PROGRAM LOAD_LASER
VAR_INPUT

END_VAR

VAR
	TMR_DELAY: TON;
	TMR1:TON;
	TMR_STOPPER_A: TON;
	TMR_STOPPER_B: TON;
END_VAR

CASE SORTER_VAR.I_CASE OF
0: //standby near lotbox
	IF SORTER_VAR.ACTIVE_ID=6 THEN
		SORTER_VAR.ACTIVE_ID:=1;
	END_IF
	CASE SORTER_VAR.I_CURRENT_TRANSACTION.TRANSPORT_INDEX OF
		2 : LASER_MOVE(STEP_DATA_1:=SORTER_VAR.I_CURRENT_TRANSACTION.STATION_NUMBER_LOAD,
				STEP_DATA_2:=3,
				STEP_DATA_3:=SORTER_VAR.I_CURRENT_TRANSACTION.JIG_INDEX_LOAD,
				STEP_DATA_4:=0,
				STEP_DATA_5:=1);
				SORTER_VAR.O_STOPPER_TRANSFER_B:=FALSE;
		1 : LASER_MOVE(STEP_DATA_1:=SORTER_VAR.I_CURRENT_TRANSACTION.STATION_NUMBER_LOAD,
				STEP_DATA_2:=3,
				STEP_DATA_3:=SORTER_VAR.I_CURRENT_TRANSACTION.JIG_INDEX_LOAD,
				STEP_DATA_4:=1,
				STEP_DATA_5:=0);
				SORTER_VAR.O_STOPPER_TRANSFER_A:=FALSE;
	END_CASE			
	SORTER_VAR.O_VACUUM_On:=FALSE;
	SORTER_VAR.O_VACUUM_OFF:=FALSE;	
	
			
1: //standby near lotbox
	
	IF SORTER_VAR.ACTIVE_ID=6 THEN
		SORTER_VAR.ACTIVE_ID:=1;
	END_IF
		LASER_MOVE(STEP_DATA_1:=SORTER_VAR.I_CURRENT_TRANSACTION.STATION_NUMBER_LOAD,
				STEP_DATA_2:=4,
				STEP_DATA_3:=SORTER_VAR.I_CURRENT_TRANSACTION.JIG_INDEX_LOAD,
				STEP_DATA_4:=0,
				STEP_DATA_5:=0);

		CASE SORTER_VAR.I_CURRENT_TRANSACTION.TRANSPORT_INDEX OF
		1:
			SORTER_VAR.I_LOADING_DONE_A:=FALSE;
		
		2:
			SORTER_VAR.I_LOADING_DONE_B:=FALSE;
	END_CASE
	
				
2://vacuum position 
	IF SORTER_VAR.ACTIVE_ID=6 THEN
		SORTER_VAR.ACTIVE_ID:=1;
	END_IF
	SORTER_VAR.I_CASE:=SORTER_VAR.I_CASE+1;
	(*LASER_MOVE(STEP_DATA_1:=SORTER_VAR.I_CURRENT_TRANSACTION.STATION_NUMBER_LOAD,
				STEP_DATA_2:=4,
				STEP_DATA_3:=SORTER_VAR.I_CURRENT_TRANSACTION.JIG_INDEX_LOAD,
				STEP_DATA_4:=0,
				STEP_DATA_5:=0);
	IF SORTER_VAR.ACTIVE_ID=3 THEN
		SORTER_VAR.O_VACUUM_ON:=TRUE;
		SORTER_VAR.O_VACUUM_OFF:=FALSE;	
	END_IF
	*)

3://vacuum position 
	IF SORTER_VAR.ACTIVE_ID=6 THEN
		SORTER_VAR.ACTIVE_ID:=1; 
	END_IF
	SORTER_VAR.I_CASE:=SORTER_VAR.I_CASE+1;
(*
		LASER_MOVE(STEP_DATA_1:=SORTER_VAR.I_CURRENT_TRANSACTION.STATION_NUMBER_LOAD,
				STEP_DATA_2:=4,
				STEP_DATA_3:=SORTER_VAR.I_CURRENT_TRANSACTION.JIG_INDEX_LOAD,
				STEP_DATA_4:=0,
				STEP_DATA_5:=0);
*)
4://vacuum position 
	IF SORTER_VAR.ACTIVE_ID=6 THEN
		SORTER_VAR.ACTIVE_ID:=1;
	END_IF
	SORTER_VAR.O_VACUUM_ON:=TRUE;
	SORTER_VAR.O_VACUUM_OFF:=FALSE;
	//CHECK JIG LASER PRESENCE	
LASER_MOVE(STEP_DATA_1:=SORTER_VAR.I_CURRENT_TRANSACTION.STATION_NUMBER_LOAD,
				STEP_DATA_2:=4,
				STEP_DATA_3:=SORTER_VAR.I_CURRENT_TRANSACTION.JIG_INDEX_LOAD,
				STEP_DATA_4:=0,
				STEP_DATA_5:=0);
(*		
	IF  SORTER_VAR.O_VACUUM_ON THEN
		TMR1(IN:=TRUE,PT:=T#2S);
		IF TMR1.Q THEN
			IF  SORTER_VAR.I_VACUUM_ON AND SORTER_VAR.O_VACUUM_ON THEN
				SORTER_VAR.JIG_LASER_PRESENCE :=TRUE;
				
				LASER_MOVE(STEP_DATA_1:=7,
				STEP_DATA_2:=4,
				STEP_DATA_3:=SORTER_VAR.I_CURRENT_TRANSACTION.JIG_INDEX_LOAD,
				STEP_DATA_4:=0,
				STEP_DATA_5:=0);
			ELSE
				SORTER_VAR.JIG_LASER_PRESENCE :=FALSE;	
				LASER_MOVE(STEP_DATA_1:=SORTER_VAR.I_CURRENT_TRANSACTION.STATION_NUMBER_LOAD,
				STEP_DATA_2:=2,
				STEP_DATA_3:=SORTER_VAR.I_CURRENT_TRANSACTION.JIG_INDEX_LOAD,
				STEP_DATA_4:=0,
				STEP_DATA_5:=0);
				
				LASER_MOVE(STEP_DATA_1:=SORTER_VAR.I_CURRENT_TRANSACTION.STATION_NUMBER_LOAD,
				STEP_DATA_2:=1,
				STEP_DATA_3:=SORTER_VAR.I_CURRENT_TRANSACTION.JIG_INDEX_LOAD,
				STEP_DATA_4:=0,
				STEP_DATA_5:=0);
				
				TMR_DELAY(IN:=TRUE,PT:=T#2S);
				IF TMR_DELAY.Q THEN
					FLAG_VAR.ALLOW_EXECUTE_LOAD_LASER:=FALSE;
					SORTER_VAR.I_CURRENT_TRANSACTION.JIG_INDEX_LOAD:=SORTER_VAR.I_CURRENT_TRANSACTION.JIG_INDEX_LOAD+0;
					SORTER_VAR.I_CASE:=0;
					TMR1(IN:=FALSE);
					SORTER_VAR.O_VACUUM_ON:=FALSE;
					SORTER_VAR.O_VACUUM_OFF:=FALSE;
				END_IF
			END_IF
		END_IF 
	END_IF
*)
				

5://vacuum position 
	IF SORTER_VAR.ACTIVE_ID=6 THEN
		SORTER_VAR.ACTIVE_ID:=1;
	END_IF

	LASER_MOVE(STEP_DATA_1:=SORTER_VAR.I_CURRENT_TRANSACTION.STATION_NUMBER_LOAD,//9,
				STEP_DATA_2:=2,
				STEP_DATA_3:=SORTER_VAR.I_CURRENT_TRANSACTION.JIG_INDEX_LOAD,
				STEP_DATA_4:=0,
				STEP_DATA_5:=0);

6://gripping position
	IF SORTER_VAR.ACTIVE_ID=6 THEN
		SORTER_VAR.ACTIVE_ID:=1;
	END_IF

	LASER_MOVE(STEP_DATA_1:=SORTER_VAR.I_CURRENT_TRANSACTION.TRANSPORT_INDEX+5,
				STEP_DATA_2:=1,
				STEP_DATA_3:=12,
				STEP_DATA_4:=0,
				STEP_DATA_5:=0);


7://placing onto LASER transport
	IF SORTER_VAR.ACTIVE_ID=6 THEN
		SORTER_VAR.ACTIVE_ID:=1;
	END_IF
	LASER_MOVE(STEP_DATA_1:=SORTER_VAR.I_CURRENT_TRANSACTION.TRANSPORT_INDEX+5,
				STEP_DATA_2:=1,
				STEP_DATA_3:=11,
				STEP_DATA_4:=0,
				STEP_DATA_5:=0);

8://placing onto LASER transport
	IF SORTER_VAR.ACTIVE_ID=6 THEN
		SORTER_VAR.ACTIVE_ID:=1;
	END_IF
	
	LASER_MOVE(STEP_DATA_1:=SORTER_VAR.I_CURRENT_TRANSACTION.TRANSPORT_INDEX+5,
				STEP_DATA_2:=1,
				STEP_DATA_3:=11,
				STEP_DATA_4:=0,
				STEP_DATA_5:=0);
	(*IF SORTER_VAR.ACTIVE_ID=3 THEN
		SORTER_VAR.O_VACUUM_On:=FALSE;
		SORTER_VAR.O_VACUUM_OFF:=TRUE;	
	END_IF
	*)
	
9://homing
	IF SORTER_VAR.ACTIVE_ID=6 THEN
		SORTER_VAR.ACTIVE_ID:=1;
	END_IF
	
			LASER_MOVE(STEP_DATA_1:=SORTER_VAR.I_CURRENT_TRANSACTION.TRANSPORT_INDEX+5,
				STEP_DATA_2:=0,
				STEP_DATA_3:=11,
				STEP_DATA_4:=0,
				STEP_DATA_5:=0);
	(*
	IF SORTER_VAR.I_VACUUM_ON THEN
		LASER_MOVE(STEP_DATA_1:=SORTER_VAR.I_CURRENT_TRANSACTION.TRANSPORT_INDEX+5,
				STEP_DATA_2:=1,
				STEP_DATA_3:=11,
				STEP_DATA_4:=0,
				STEP_DATA_5:=0);
	ELSE
		SORTER_VAR.O_VACUUM_On:=FALSE;
		SORTER_VAR.O_VACUUM_OFF:=TRUE;
	END_IF	
	*)			
10://pusH LASER transport
	IF SORTER_VAR.ACTIVE_ID=6 THEN
		SORTER_VAR.ACTIVE_ID:=1;
	END_IF
	SORTER_VAR.O_VACUUM_OFF:=FALSE;
	CASE SORTER_VAR.I_CURRENT_TRANSACTION.TRANSPORT_INDEX OF
		2 :
			IF NOT SORTER_VAR.I_LASER_TRANSFER_AT_FRONT_B THEN
				LASER_MOVE(STEP_DATA_1:=0,
				STEP_DATA_2:=0,
				STEP_DATA_3:=0,
				STEP_DATA_4:=0,
				STEP_DATA_5:=2);
			END_IF
				 
		1 : 
			IF NOT SORTER_VAR.I_LASER_TRANSFER_AT_FRONT_A THEN
				LASER_MOVE(STEP_DATA_1:=0,
				STEP_DATA_2:=0,
				STEP_DATA_3:=0,
				STEP_DATA_4:=2,
				STEP_DATA_5:=0);
			END_IF
	END_CASE			 
11:
				CASE SORTER_VAR.I_CURRENT_TRANSACTION.TRANSPORT_INDEX OF
		1:	
			//IF SORTER_VAR.I_LASER_TRANSFER_AT_FRONT_A THEN
				
				TMR_STOPPER_A(IN:=TRUE,PT:=T#0.8S);
				IF TMR_STOPPER_A.Q THEN
					SORTER_VAR.O_STOPPER_TRANSFER_A:=TRUE;
					SORTER_VAR.I_LOADING_DONE_A:=TRUE;
					TMR1(IN:=FALSE);
	TMR_DELAY(IN:=FALSE);
	FLAG_VAR.ALLOW_EXECUTE_LOAD_LASER:=FALSE;	
					SORTER_VAR.I_CASE:=100;
						SORTER_VAR.O_VACUUM_On:=FALSE;
	SORTER_VAR.O_VACUUM_OFF:=FALSE;
	
END_IF
				
(*			ELSE
				TMR_STOPPER_A(IN:=FALSE);
				LASER_MOVE(STEP_DATA_1:=0,
				STEP_DATA_2:=0,
				STEP_DATA_3:=0,
				STEP_DATA_4:=2,
				STEP_DATA_5:=0);
			END_IF
*)			
			2:
			//IF SORTER_VAR.I_LASER_TRANSFER_AT_FRONT_B THEN
				
				TMR_STOPPER_B(IN:=TRUE,PT:=T#0.8S);
				IF TMR_STOPPER_B.Q THEN
					SORTER_VAR.O_STOPPER_TRANSFER_B:=TRUE;	
					SORTER_VAR.I_LOADING_DONE_B:=TRUE;
					TMR1(IN:=FALSE);
	TMR_DELAY(IN:=FALSE);
	FLAG_VAR.ALLOW_EXECUTE_LOAD_LASER:=FALSE;	
					SORTER_VAR.I_CASE:=100;
						SORTER_VAR.O_VACUUM_On:=FALSE;
	SORTER_VAR.O_VACUUM_OFF:=FALSE;
			END_IF
(*			ELSE
				TMR_STOPPER_B(IN:=FALSE);
				LASER_MOVE(STEP_DATA_1:=0,
				STEP_DATA_2:=0,
				STEP_DATA_3:=0,
				STEP_DATA_4:=0,
				STEP_DATA_5:=2);
			END_IF
*)			
	END_CASE
100:
	SORTER_VAR.O_VACUUM_On:=FALSE;
	SORTER_VAR.O_VACUUM_OFF:=FALSE;
	TMR1(IN:=FALSE);
	TMR_DELAY(IN:=FALSE);
	FLAG_VAR.ALLOW_EXECUTE_LOAD_LASER:=FALSE;								
								
END_CASE

END_PROGRAM

(* stored: Version 1.1.0.1, ProductVersion 3.1.4020.12
   POU LOAD_LASER: Id {ed8e2b66-0fd3-4437-8ee5-0030e16f334b}, SpecialFunc None *)
